TYPE TcoCylinderConfig :
STRUCT
	TimeToReachHomePosition : TIME := T#10S;
	TimeToReachWorkPosition : TIME := T#10S;
	TimeToRefill : TIME := T#1000MS;
END_STRUCT
END_TYPE

(* stored: Version 1.1.0.1
   DUT TcoCylinderConfig: Id {ab3dceba-9fd6-4308-a457-8d8ae3c511fc} *)
